# B&R Automation Studio project Fuellstand
Automation Studio 4.9.2.46; technology packages: mappView 5.12.1

## Configuration X20cp1584

CPU X20CP1584, AutomationRuntime C4.90, Build 4.1.2, Safety 0.0, Vc V4.62.0

### Hardware
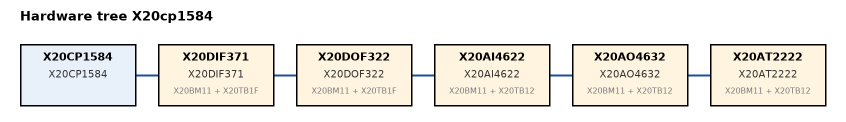
```
X20AI4622 : X20AI4622 v1.1.0.0  [SS1 -> X20TB12.SS; SL -> X20BM11b.SL1]
  LowerLimit = 0
X20AO4632 : X20AO4632 v1.1.0.0  [SS1 -> X20TB12a.SS; SL -> X20BM11c.SL1]
X20AT2222 : X20AT2222 v1.3.0.0  [SS1 -> X20TB12b.SS; SL -> X20BM11d.SL1]
X20BM11 : X20BM11 v1.0.0.1  [X2X1 -> X20CP1584.IF6]
X20BM11a : X20BM11 v1.0.0.1  [X2X1 -> X20BM11.X2X2]
X20BM11b : X20BM11 v1.0.0.1  [X2X1 -> X20BM11a.X2X2]
X20BM11c : X20BM11 v1.0.0.1  [X2X1 -> X20BM11b.X2X2]
X20BM11d : X20BM11 v1.0.0.1  [X2X1 -> X20BM11c.X2X2]
X20CP1584 : X20CP1584 v1.9.0.0
  Connector IF2:
    ActivateDevice = 1
    Mode = Manual
    InternetAddress = 10.10.4.1
  Connector IF3:
    DNAConfiguration = manual
  ConfigurationID = Fuellstand_X20cp1584
  Simulation = 1
  ActivateOpcUa = 1
  OpcUaInformationModels_PV_Version = 1
X20DIF371 : X20DIF371 v1.1.0.0  [SS1 -> X20TB1F.SS; SL -> X20BM11.SL1]
X20DOF322 : X20DOF322 v1.4.0.0  [SS1 -> X20TB1F1.SS; SL -> X20BM11a.SL1]
X20TB12 : X20TB12 v1.0.0.0
X20TB12a : X20TB12 v1.0.0.0
X20TB12b : X20TB12 v1.0.0.0
X20TB1F : X20TB1F v1.0.0.0
X20TB1F1 : X20TB1F v1.0.0.0
```

### IoMap.iom - X20CP1584/IoMap.iom
```iecst
VAR_CONFIG
	::Program:DiTankB002Leer_L002L AT %IX."X20DIF371".DigitalInput01 INVERSE;
	::Program:DoVentilAblass_Y002 AT %QX."X20DOF322".DigitalOutput01;
	::Program:AiFuellstandTank_L001 AT %IW."X20AI4622".AnalogInput01;
	::Program:AoPumpe_P001 AT %QW."X20AO4632".AnalogOutput01;
END_VAR
```

## Logical view

Binary libraries used (declarations not repeated): operator, runtime, astime, AsIecCon, standard, LoopCont 3.10.0, sys_lib, brsystem, MTBasics 5.06.0, MTTypes


### Program Logical/Program (IEC)

#### Variables.var
```iecst
VAR
	varPID_I : REAL;
	varPID_P : REAL;
	varSimulation : BOOL;
	DoVentilAblass_Y002 : BOOL;
	DiTankB002Leer_L002L : BOOL;
	AoPumpe_P001 : INT;
	varPumpe : INT;
	AiFuellstandTank_L001 : INT;
	dh : REAL;
	h : REAL;
	varFuellstandUnten : REAL;
	varFuellstandOben : REAL;
	varSollFuellstand : REAL;
	varPidEnb : BOOL; (*PID*) (*SetValue : REAL := 0.0; (* set value *) (*ActValue : REAL := 0.0; (* actual value *)
	PID : MTBasicsPID := (0); (* function block MTBasicsPID *)
	tzyk : REAL;
	Kp : REAL;
	Kr : REAL;
END_VAR
```

#### Cyclic.st
```iecst
PROGRAM _CYCLIC

	(* http://localhost:81/index.html?visuId=FirstVisu *)

	IF(varSimulation) THEN
		dh := (Kr * (1 + 2 * BOOL_TO_INT(DoVentilAblass_Y002)) * h) + (Kp * REAL_TO_INT(PID.Out) / 100);
		h := h + dh;
		varFuellstandOben := h * 100;
		varPumpe := 0;
	ELSE
		varFuellstandOben := INT_TO_REAL(AiFuellstandTank_L001) / 232.0;
		IF(DiTankB002Leer_L002L) THEN
			varPumpe := 0;
		ELSE
			varPumpe := REAL_TO_INT(PID.Out);
		END_IF
	END_IF

	IF((varSollFuellstand >= 20) AND (varSollFuellstand <= 100))THEN
		varPidEnb := TRUE;

		IF((varFuellstandOben - varSollFuellstand) >= 10.0)THEN
			DoVentilAblass_Y002 := TRUE;
		ELSE
			DoVentilAblass_Y002 := FALSE;
		END_IF
	ELSE
		varPidEnb := FALSE;
		DoVentilAblass_Y002 := TRUE;
	END_IF

	AoPumpe_P001 := varPumpe * 320;
	varFuellstandUnten := 100 - varFuellstandOben;

	(* call function block *)
	PID.SetValue := varSollFuellstand;
	PID.ActValue := varFuellstandOben;
	PID.Enable := varPidEnb;
	PID.PIDParameters.Gain := varPID_P;
	PID.PIDParameters.IntegrationTime := varPID_I;
	PID();

END_PROGRAM
```

- Hardware.hw (not shown)

#### Init.st
```iecst
PROGRAM _INIT
	(* SIMULATION *)
	varSimulation := 1;
	tzyk := 0.1;
	Kr := -0.019 * tzyk;
	Kp := 0.035 * tzyk;
	h := 0;

	(* PID parameters *)
	varPID_P := 5;
	varPID_I := 5;
	PID.PIDParameters.DerivativeTime := 0.0;
	PID.PIDParameters.FilterTime := 0.0;
	(* output limits *)
	PID.MinOut := 0;
	PID.MaxOut := 100;
	PID.Enable := FALSE;

END_PROGRAM
```

- Visualisation Logical/mappView (not shown)

Listed in the project but not available here: Logical/Global.typ, Logical/Global.var
